// Mitsubishi GX Works2 project: 프로젝트1   PLC: Q02/Q02H

PROGRAM MAIN
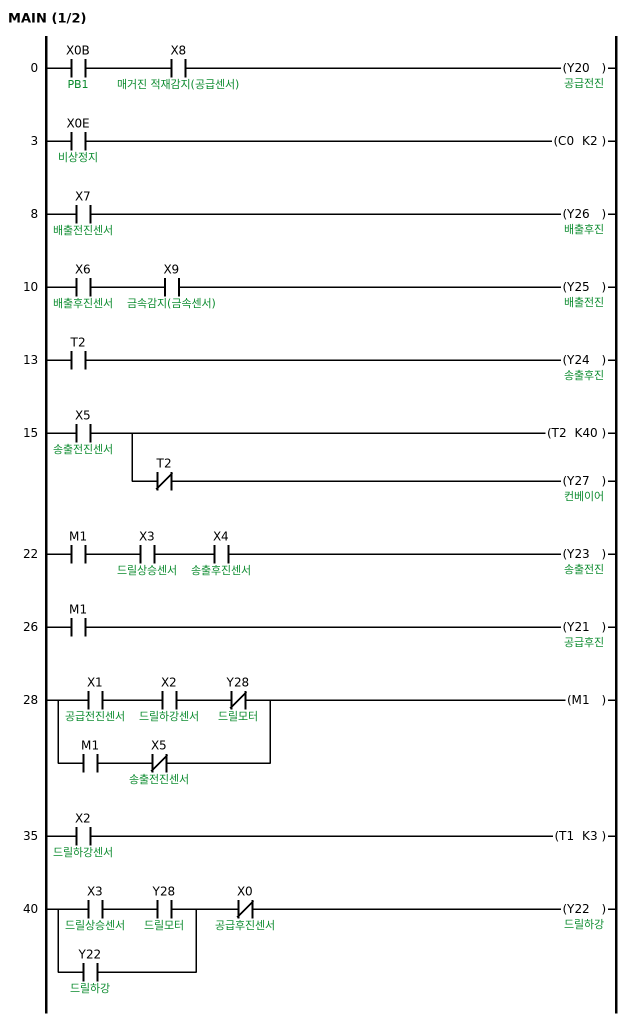
0     LD      X0B  ; PB1
      AND     X8  ; 매거진 적재감지(공급센서)
      OUT     Y20  ; 공급전진
3     LD      X0E  ; 비상정지
      OUT     C0 K2
8     LD      X7  ; 배출전진센서
      OUT     Y26  ; 배출후진
10    LD      X6  ; 배출후진센서
      AND     X9  ; 금속감지(금속센서)
      OUT     Y25  ; 배출전진
13    LD      T2
      OUT     Y24  ; 송출후진
15    LD      X5  ; 송출전진센서
      OUT     T2 K40
      ANI     T2
      OUT     Y27  ; 컨베이어
22    LD      M1
      AND     X3  ; 드릴상승센서
      AND     X4  ; 송출후진센서
      OUT     Y23  ; 송출전진
26    LD      M1
      OUT     Y21  ; 공급후진
28    LD      X1  ; 공급전진센서
      AND     X2  ; 드릴하강센서
      ANI     Y28  ; 드릴모터
      LD      M1
      ANI     X5  ; 송출전진센서
      ORB
      OUT     M1
35    LD      X2  ; 드릴하강센서
      OUT     T1 K3
40    LD      X3  ; 드릴상승센서
      AND     Y28  ; 드릴모터
      OR      Y22  ; 드릴하강
      ANI     X0  ; 공급후진센서
      OUT     Y22  ; 드릴하강
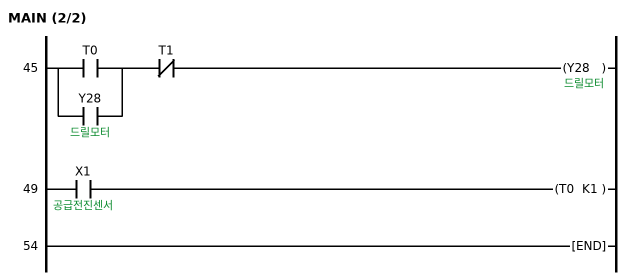
45    LD      T0
      OR      Y28  ; 드릴모터
      ANI     T1
      OUT     Y28  ; 드릴모터
49    LD      X1  ; 공급전진센서
      OUT     T0 K1
54    END
END_PROGRAM

// device comments not shown above
X0A  ; 비금속 감지(가공센서)
X0C  ; PB2
X0D  ; PB3
Y29  ; 적색램프
Y2A  ; 황색램프
Y2B  ; 녹색램프
